// This function has been automatically generated from the project information.
{attribute 'signature_flag' := '1073741824'}
{attribute 'TcGenerated'}
{attribute 'no-analysis'}
FUNCTION F_GetVersion : ST_LibVersion
VAR_INPUT
	
END_VAR

F_GetVersion.iMajor := 4;
F_GetVersion.iMinor := 0;
F_GetVersion.iBuild := 0;
F_GetVersion.iRevision := 1;
F_GetVersion.sVersion := '4.0.0.1';
F_GetVersion.nFlags := 0;

END_FUNCTION

(* stored: Version 1.1.0.1, ProductVersion 3.1.4026.8
   POU F_GetVersion: Id {7a367244-f92d-433f-88d7-35d85292607e}, SpecialFunc None *)
